LIN {X 0,Y 71.965,Z 1200.65,A -85,B 0,C 180,E1 3862.817,E2 3862.817} C_VEL
LIN {X 0,Y 71.914,Z 1200.39,A -85,B 0,C 180,E1 3872.39,E2 3872.39} C_VEL
LIN {X 0,Y 72.406,Z 1199.456,A -85,B 0,C 180,E1 3884.392,E2 3884.392} C_VEL
LIN {X 0,Y 75.878,Z 1197.57,A -85,B 0,C 180,E1 3899.18,E2 3899.18} C_VEL
LIN {X 0,Y 84.039,Z 1194.488,A -85,B 0,C 180,E1 3913.634,E2 3913.634} C_VEL
LIN {X 0,Y 99.563,Z 1189.174,A -85,B 0,C 180,E1 3927.841,E2 3927.841} C_VEL
LIN {X 0,Y 118.686,Z 1182.09,A -85,B 0,C 180,E1 3937.923,E2 3937.923} C_VEL
LIN {X 0,Y 136.218,Z 1175.067,A -85,B 0,C 180,E1 3944.061,E2 3944.061} C_VEL
LIN {X 0,Y 154.904,Z 1166.814,A -85,B 0,C 180,E1 3948.846,E2 3948.846} C_VEL
LIN {X 0,Y 178.199,Z 1155.352,A -85,B 0,C 180,E1 3953.279,E2 3953.279} C_VEL
LIN {X 0,Y 200.35,Z 1142.821,A -85,B 0,C 180,E1 3956.476,E2 3956.476} C_VEL
LIN {X 0,Y 219.029,Z 1131.127,A -85,B 0,C 180,E1 3958.647,E2 3958.647} C_VEL
LIN {X 0,Y 236.971,Z 1118.762,A -85,B 0,C 180,E1 3960.395,E2 3960.395} C_VEL
LIN {X 0,Y 256.541,Z 1103.89,A -85,B 0,C 180,E1 3962.01,E2 3962.01} C_VEL
LIN {X 0,Y 279.003,Z 1084.625,A -85,B 0,C 180,E1 3963.579,E2 3963.579} C_VEL
LIN {X 0,Y 280.373,Z 1083.351,A -85,B 0,C 180,E1 3963.668,E2 3963.668} C_VEL
LIN {X 0,Y 271.689,Z 1091.139,A -85,B 0,C 180,E1 3964.25,E2 3964.25} C_VEL
LIN {X 0,Y 266.605,Z 1095.454,A -85,B 0,C 180,E1 3964.415,E2 3964.415} C_VEL
LIN {X 0,Y 259.732,Z 1101.256,A -85,B 0,C 180,E1 3964.211,E2 3964.211} C_VEL
LIN {X 0,Y 244.077,Z 1113.399,A -85,B 0,C 180,E1 3962.959,E2 3962.959} C_VEL
LIN {X 0,Y 220.956,Z 1129.444,A -85,B 0,C 180,E1 3961.037,E2 3961.037} C_VEL
LIN {X 0,Y 201.994,Z 1141.263,A -85,B 0,C 180,E1 3959.115,E2 3959.115} C_VEL
LIN {X 0,Y 182.28,Z 1152.355,A -85,B 0,C 180,E1 3956.678,E2 3956.678} C_VEL
LIN {X 0,Y 158.208,Z 1164.433,A -85,B 0,C 180,E1 3952.849,E2 3952.849} C_VEL
LIN {X 0,Y 135.95,Z 1174.072,A -85,B 0,C 180,E1 3948.003,E2 3948.003} C_VEL
LIN {X 0,Y 117.478,Z 1181.227,A -85,B 0,C 180,E1 3942.408,E2 3942.408} C_VEL
LIN {X 0,Y 100.411,Z 1187.206,A -85,B 0,C 180,E1 3934.977,E2 3934.977} C_VEL
LIN {X 0,Y 83.535,Z 1192.691,A -85,B 0,C 180,E1 3923.315,E2 3923.315} C_VEL
LIN {X 0,Y 69.868,Z 1197.075,A -85,B 0,C 180,E1 3904.919,E2 3904.919} C_VEL
LIN {X 0,Y 64.688,Z 1199.265,A -85,B 0,C 180,E1 3887.078,E2 3887.078} C_VEL
LIN {X 0,Y 63.912,Z 1200.269,A -85,B 0,C 180,E1 3873.588,E2 3873.588} C_VEL
LIN {X 0,Y 63.942,Z 1200.51,A -85,B 0,C 180,E1 3863.716,E2 3863.716} C_VEL
LIN {X 0,Y 65.136,Z 1200.516,A -85,B 0,C 180,E1 3850.263,E2 3850.263} C_VEL
LIN {X 0,Y 71.141,Z 1199.657,A -85,B 0,C 180,E1 3832.818,E2 3832.818} C_VEL
LIN {X 0,Y 82.509,Z 1197.706,A -85,B 0,C 180,E1 3818.031,E2 3818.031} C_VEL
LIN {X 0,Y 97.644,Z 1194.686,A -85,B 0,C 180,E1 3807.018,E2 3807.018} C_VEL
LIN {X 0,Y 116.093,Z 1190.376,A -85,B 0,C 180,E1 3798.669,E2 3798.669} C_VEL
LIN {X 0,Y 140.962,Z 1183.473,A -85,B 0,C 180,E1 3791.456,E2 3791.456} C_VEL
LIN {X 0,Y 165.113,Z 1175.312,A -85,B 0,C 180,E1 3786.726,E2 3786.726} C_VEL
LIN {X 0,Y 186.353,Z 1167.079,A -85,B 0,C 180,E1 3783.661,E2 3783.661} C_VEL
LIN {X 0,Y 190.059,Z 1165.559,A -85,B 0,C 180,E1 3783.17,E2 3783.17} C_VEL
LIN {X 0,Y 167.976,Z 1174.095,A -85,B 0,C 180,E1 3780.074,E2 3780.074} C_VEL
LIN {X 0,Y 147.292,Z 1181.068,A -85,B 0,C 180,E1 3776.262,E2 3776.262} C_VEL
LIN {X 0,Y 125.611,Z 1187.374,A -85,B 0,C 180,E1 3770.762,E2 3770.762} C_VEL
LIN {X 0,Y 101.386,Z 1193.141,A -85,B 0,C 180,E1 3761.217,E2 3761.217} C_VEL
LIN {X 0,Y 85.017,Z 1196.305,A -85,B 0,C 180,E1 3750.398,E2 3750.398} C_VEL
LIN {X 0,Y 73.034,Z 1198.239,A -85,B 0,C 180,E1 3736.518,E2 3736.518} C_VEL
LIN {X 0,Y 66.274,Z 1199.108,A -85,B 0,C 180,E1 3720.686,E2 3720.686} C_VEL
LIN {X 0,Y 64.065,Z 1199.187,A -85,B 0,C 180,E1 3705.386,E2 3705.386} C_VEL
LIN {X 0,Y 63.918,Z 1198.899,A -85,B 0,C 180,E1 3694.486,E2 3694.486} C_VEL
LIN {X 0,Y 64.676,Z 1197.981,A -85,B 0,C 180,E1 3681.107,E2 3681.107} C_VEL
LIN {X 0,Y 69.216,Z 1196.076,A -85,B 0,C 180,E1 3664.319,E2 3664.319} C_VEL
LIN {X 0,Y 80.178,Z 1192.658,A -85,B 0,C 180,E1 3647.67,E2 3647.67} C_VEL
LIN {X 0,Y 99.235,Z 1186.688,A -85,B 0,C 180,E1 3633.251,E2 3633.251} C_VEL
LIN {X 0,Y 116.37,Z 1180.839,A -85,B 0,C 180,E1 3625.556,E2 3625.556} C_VEL
LIN {X 0,Y 134.074,Z 1174.148,A -85,B 0,C 180,E1 3620.009,E2 3620.009} C_VEL
LIN {X 0,Y 152.684,Z 1166.317,A -85,B 0,C 180,E1 3615.712,E2 3615.712} C_VEL
LIN {X 0,Y 175.646,Z 1155.489,A -85,B 0,C 180,E1 3611.735,E2 3611.735} C_VEL
LIN {X 0,Y 199.228,Z 1142.62,A -85,B 0,C 180,E1 3608.632,E2 3608.632} C_VEL
LIN {X 0,Y 218.421,Z 1130.906,A -85,B 0,C 180,E1 3606.612,E2 3606.612} C_VEL
LIN {X 0,Y 236.861,Z 1118.458,A -85,B 0,C 180,E1 3604.985,E2 3604.985} C_VEL
LIN {X 0,Y 253.944,Z 1105.754,A -85,B 0,C 180,E1 3603.68,E2 3603.68} C_VEL
LIN {X 0,Y 244.077,Z 1113.399,A -85,B 0,C 180,E1 3602.959,E2 3602.959} C_VEL
LIN {X 0,Y 237.846,Z 1117.949,A -85,B 0,C 180,E1 3602.729,E2 3602.729} C_VEL
LIN {X 0,Y 221.123,Z 1129.147,A -85,B 0,C 180,E1 3602.95,E2 3602.95} C_VEL
LIN {X 0,Y 214.651,Z 1133.273,A -85,B 0,C 180,E1 3602.675,E2 3602.675} C_VEL
LIN {X 0,Y 188.973,Z 1148.299,A -85,B 0,C 180,E1 3600.154,E2 3600.154} C_VEL
LIN {X 0,Y 168.131,Z 1158.981,A -85,B 0,C 180,E1 3597.538,E2 3597.538} C_VEL
LIN {X 0,Y 148.685,Z 1167.89,A -85,B 0,C 180,E1 3594.412,E2 3594.412} C_VEL
LIN {X 0,Y 128.635,Z 1176.071,A -85,B 0,C 180,E1 3590.154,E2 3590.154} C_VEL
LIN {X 0,Y 104.718,Z 1184.631,A -85,B 0,C 180,E1 3582.708,E2 3582.708} C_VEL
LIN {X 0,Y 84.953,Z 1190.695,A -85,B 0,C 180,E1 3572.676,E2 3572.676} C_VEL
LIN {X 0,Y 70.5,Z 1194.813,A -85,B 0,C 180,E1 3559.982,E2 3559.982} C_VEL
LIN {X 0,Y 60.889,Z 1197.634,A -85,B 0,C 180,E1 3543.939,E2 3543.939} C_VEL
LIN {X 0,Y 56.552,Z 1199.355,A -85,B 0,C 180,E1 3526.432,E2 3526.432} C_VEL
LIN {X 0,Y 55.914,Z 1200.217,A -85,B 0,C 180,E1 3512.049,E2 3512.049} C_VEL
LIN {X 0,Y 56.076,Z 1200.473,A -85,B 0,C 180,E1 3499.729,E2 3499.729} C_VEL
LIN {X 0,Y 59.309,Z 1200.261,A -85,B 0,C 180,E1 3480.732,E2 3480.732} C_VEL
LIN {X 0,Y 69.759,Z 1198.932,A -85,B 0,C 180,E1 3461.249,E2 3461.249} C_VEL
LIN {X 0,Y 90.166,Z 1195.477,A -85,B 0,C 180,E1 3444.591,E2 3444.591} C_VEL
LIN {X 0,Y 110.166,Z 1191.213,A -85,B 0,C 180,E1 3435.835,E2 3435.835} C_VEL
LIN {X 0,Y 130.019,Z 1186.162,A -85,B 0,C 180,E1 3430.158,E2 3430.158} C_VEL
LIN {X 0,Y 151.755,Z 1179.668,A -85,B 0,C 180,E1 3425.798,E2 3425.798} C_VEL
LIN {X 0,Y 168.931,Z 1173.751,A -85,B 0,C 180,E1 3423.16,E2 3423.16} C_VEL
LIN {X 0,Y 147.979,Z 1180.695,A -85,B 0,C 180,E1 3419.861,E2 3419.861} C_VEL
LIN {X 0,Y 126.42,Z 1186.819,A -85,B 0,C 180,E1 3415.231,E2 3415.231} C_VEL
LIN {X 0,Y 101.539,Z 1192.672,A -85,B 0,C 180,E1 3407.124,E2 3407.124} C_VEL
LIN {X 0,Y 81.149,Z 1196.331,A -85,B 0,C 180,E1 3395.751,E2 3395.751} C_VEL
LIN {X 0,Y 67.433,Z 1198.295,A -85,B 0,C 180,E1 3381.8,E2 3381.8} C_VEL
LIN {X 0,Y 59.247,Z 1199.184,A -85,B 0,C 180,E1 3365.015,E2 3365.015} C_VEL
LIN {X 0,Y 56.185,Z 1199.288,A -85,B 0,C 180,E1 3347.61,E2 3347.61} C_VEL
LIN {X 0,Y 55.918,Z 1198.999,A -85,B 0,C 180,E1 3335.13,E2 3335.13} C_VEL
LIN {X 0,Y 56.651,Z 1198.169,A -85,B 0,C 180,E1 3320.86,E2 3320.86} C_VEL
LIN {X 0,Y 60.95,Z 1196.554,A -85,B 0,C 180,E1 3303.71,E2 3303.71} C_VEL
LIN {X 0,Y 70.256,Z 1193.919,A -85,B 0,C 180,E1 3288.019,E2 3288.019} C_VEL
LIN {X 0,Y 83.774,Z 1190.178,A -85,B 0,C 180,E1 3275.748,E2 3275.748} C_VEL
LIN {X 0,Y 100.605,Z 1185.167,A -85,B 0,C 180,E1 3266.562,E2 3266.562} C_VEL
LIN {X 0,Y 123.517,Z 1177.516,A -85,B 0,C 180,E1 3258.719,E2 3258.719} C_VEL
LIN {X 0,Y 147.354,Z 1168.034,A -85,B 0,C 180,E1 3253.339,E2 3253.339} C_VEL
LIN {X 0,Y 166.592,Z 1159.398,A -85,B 0,C 180,E1 3250.167,E2 3250.167} C_VEL
LIN {X 0,Y 186.601,Z 1149.342,A -85,B 0,C 180,E1 3247.574,E2 3247.574} C_VEL
LIN {X 0,Y 209.829,Z 1136.257,A -85,B 0,C 180,E1 3245.189,E2 3245.189} C_VEL
LIN {X 0,Y 227.229,Z 1125.213,A -85,B 0,C 180,E1 3243.69,E2 3243.69} C_VEL
LIN {X 0,Y 214.651,Z 1133.273,A -85,B 0,C 180,E1 3242.675,E2 3242.675} C_VEL
LIN {X 0,Y 208.11,Z 1137.331,A -85,B 0,C 180,E1 3242.378,E2 3242.378} C_VEL
LIN {X 0,Y 189.592,Z 1147.773,A -85,B 0,C 180,E1 3242.522,E2 3242.522} C_VEL
LIN {X 0,Y 183.785,Z 1150.764,A -85,B 0,C 180,E1 3242.181,E2 3242.181} C_VEL
LIN {X 0,Y 163.976,Z 1160.546,A -85,B 0,C 180,E1 3239.922,E2 3239.922} C_VEL
LIN {X 0,Y 139.286,Z 1171.34,A -85,B 0,C 180,E1 3236.198,E2 3236.198} C_VEL
LIN {X 0,Y 114.458,Z 1180.427,A -85,B 0,C 180,E1 3230.793,E2 3230.793} C_VEL
LIN {X 0,Y 95.414,Z 1186.509,A -85,B 0,C 180,E1 3224.597,E2 3224.597} C_VEL
LIN {X 0,Y 77.874,Z 1191.456,A -85,B 0,C 180,E1 3215.727,E2 3215.727} C_VEL
LIN {X 0,Y 61.649,Z 1195.633,A -85,B 0,C 180,E1 3201.122,E2 3201.122} C_VEL
LIN {X 0,Y 50.064,Z 1198.813,A -85,B 0,C 180,E1 3176.064,E2 3176.064} C_VEL
LIN {X 0,Y 47.932,Z 1199.998,A -85,B 0,C 180,E1 3155.987,E2 3155.987} C_VEL
LIN {X 0,Y 47.918,Z 1200.25,A -85,B 0,C 180,E1 3145.212,E2 3145.212} C_VEL
LIN {X 0,Y 49.613,Z 1200.409,A -85,B 0,C 180,E1 3126.23,E2 3126.23} C_VEL
LIN {X 0,Y 58.849,Z 1199.542,A -85,B 0,C 180,E1 3103.065,E2 3103.065} C_VEL
LIN {X 0,Y 73.954,Z 1197.556,A -85,B 0,C 180,E1 3087.367,E2 3087.367} C_VEL
LIN {X 0,Y 92.135,Z 1194.501,A -85,B 0,C 180,E1 3077.257,E2 3077.257} C_VEL
LIN {X 0,Y 112.986,Z 1190.146,A -85,B 0,C 180,E1 3070.195,E2 3070.195} C_VEL
LIN {X 0,Y 139.408,Z 1183.343,A -85,B 0,C 180,E1 3064.492,E2 3064.492} C_VEL
LIN {X 0,Y 147.603,Z 1180.812,A -85,B 0,C 180,E1 3063.158,E2 3063.158} C_VEL
LIN {X 0,Y 125.994,Z 1186.779,A -85,B 0,C 180,E1 3059.2,E2 3059.2} C_VEL
LIN {X 0,Y 100.889,Z 1192.515,A -85,B 0,C 180,E1 3052.329,E2 3052.329} C_VEL
LIN {X 0,Y 77.993,Z 1196.366,A -85,B 0,C 180,E1 3041.561,E2 3041.561} C_VEL
LIN {X 0,Y 62.498,Z 1198.353,A -85,B 0,C 180,E1 3027.985,E2 3027.985} C_VEL
LIN {X 0,Y 52.181,Z 1199.284,A -85,B 0,C 180,E1 3009.222,E2 3009.222} C_VEL
LIN {X 0,Y 48.289,Z 1199.365,A -85,B 0,C 180,E1 2989.347,E2 2989.347} C_VEL
LIN {X 0,Y 47.916,Z 1199.075,A -85,B 0,C 180,E1 2974.788,E2 2974.788} C_VEL
LIN {X 0,Y 48.918,Z 1198.224,A -85,B 0,C 180,E1 2958.206,E2 2958.206} C_VEL
LIN {X 0,Y 54.283,Z 1196.588,A -85,B 0,C 180,E1 2938.953,E2 2938.953} C_VEL
LIN {X 0,Y 65.167,Z 1193.919,A -85,B 0,C 180,E1 2922.464,E2 2922.464} C_VEL
LIN {X 0,Y 80.863,Z 1189.966,A -85,B 0,C 180,E1 2910.056,E2 2910.056} C_VEL
LIN {X 0,Y 101.174,Z 1184.247,A -85,B 0,C 180,E1 2900.842,E2 2900.842} C_VEL
LIN {X 0,Y 126.644,Z 1175.714,A -85,B 0,C 180,E1 2893.812,E2 2893.812} C_VEL
LIN {X 0,Y 147.206,Z 1167.691,A -85,B 0,C 180,E1 2889.98,E2 2889.98} C_VEL
LIN {X 0,Y 167.276,Z 1158.818,A -85,B 0,C 180,E1 2887.148,E2 2887.148} C_VEL
LIN {X 0,Y 188.633,Z 1148.176,A -85,B 0,C 180,E1 2884.795,E2 2884.795} C_VEL
LIN {X 0,Y 200.192,Z 1141.797,A -85,B 0,C 180,E1 2883.723,E2 2883.723} C_VEL
LIN {X 0,Y 183.785,Z 1150.764,A -85,B 0,C 180,E1 2882.181,E2 2882.181} C_VEL
LIN {X 0,Y 176.956,Z 1154.326,A -85,B 0,C 180,E1 2881.79,E2 2881.79} C_VEL
LIN {X 0,Y 157.694,Z 1163.257,A -85,B 0,C 180,E1 2881.861,E2 2881.861} C_VEL
LIN {X 0,Y 151.662,Z 1165.78,A -85,B 0,C 180,E1 2881.42,E2 2881.42} C_VEL
LIN {X 0,Y 130.041,Z 1174.353,A -85,B 0,C 180,E1 2878.26,E2 2878.26} C_VEL
LIN {X 0,Y 109.563,Z 1181.432,A -85,B 0,C 180,E1 2874.109,E2 2874.109} C_VEL
LIN {X 0,Y 87.756,Z 1187.944,A -85,B 0,C 180,E1 2867.497,E2 2867.497} C_VEL
LIN {X 0,Y 64.203,Z 1193.815,A -85,B 0,C 180,E1 2854.589,E2 2854.589} C_VEL
LIN {X 0,Y 49.212,Z 1197.11,A -85,B 0,C 180,E1 2837.005,E2 2837.005} C_VEL
LIN {X 0,Y 41.445,Z 1199.042,A -85,B 0,C 180,E1 2814.212,E2 2814.212} C_VEL
LIN {X 0,Y 39.912,Z 1199.997,A -85,B 0,C 180,E1 2794.31,E2 2794.31} C_VEL
LIN {X 0,Y 39.993,Z 1200.193,A -85,B 0,C 180,E1 2781.373,E2 2781.373} C_VEL
LIN {X 0,Y 43.269,Z 1200.255,A -85,B 0,C 180,E1 2757.894,E2 2757.894} C_VEL
LIN {X 0,Y 54.873,Z 1199.344,A -85,B 0,C 180,E1 2734.92,E2 2734.92} C_VEL
LIN {X 0,Y 71.607,Z 1197.369,A -85,B 0,C 180,E1 2720.687,E2 2720.687} C_VEL
LIN {X 0,Y 90.923,Z 1194.328,A -85,B 0,C 180,E1 2711.843,E2 2711.843} C_VEL
LIN {X 0,Y 113.523,Z 1189.789,A -85,B 0,C 180,E1 2705.586,E2 2705.586} C_VEL
LIN {X 0,Y 125.913,Z 1186.804,A -85,B 0,C 180,E1 2703.135,E2 2703.135} C_VEL
LIN {X 0,Y 99.535,Z 1192.619,A -85,B 0,C 180,E1 2697.121,E2 2697.121} C_VEL
LIN {X 0,Y 74.815,Z 1196.513,A -85,B 0,C 180,E1 2687.317,E2 2687.317} C_VEL
LIN {X 0,Y 57.574,Z 1198.486,A -85,B 0,C 180,E1 2674.267,E2 2674.267} C_VEL
LIN {X 0,Y 45.478,Z 1199.385,A -85,B 0,C 180,E1 2654.712,E2 2654.712} C_VEL
LIN {X 0,Y 40.443,Z 1199.442,A -85,B 0,C 180,E1 2631.768,E2 2631.768} C_VEL
LIN {X 0,Y 39.918,Z 1199.174,A -85,B 0,C 180,E1 2615.75,E2 2615.75} C_VEL
LIN {X 0,Y 40.924,Z 1198.412,A -85,B 0,C 180,E1 2597.298,E2 2597.298} C_VEL
LIN {X 0,Y 47.08,Z 1196.843,A -85,B 0,C 180,E1 2575.012,E2 2575.012} C_VEL
LIN {X 0,Y 59.951,Z 1194.099,A -85,B 0,C 180,E1 2556.818,E2 2556.818} C_VEL
LIN {X 0,Y 76.29,Z 1190.359,A -85,B 0,C 180,E1 2545.27,E2 2545.27} C_VEL
LIN {X 0,Y 95.361,Z 1185.349,A -85,B 0,C 180,E1 2537.422,E2 2537.422} C_VEL
LIN {X 0,Y 120.232,Z 1177.7,A -85,B 0,C 180,E1 2531.101,E2 2531.101} C_VEL
LIN {X 0,Y 145.05,Z 1168.378,A -85,B 0,C 180,E1 2526.966,E2 2526.966} C_VEL
LIN {X 0,Y 165.48,Z 1159.584,A -85,B 0,C 180,E1 2524.472,E2 2524.472} C_VEL
LIN {X 0,Y 172.336,Z 1156.447,A -85,B 0,C 180,E1 2523.712,E2 2523.712} C_VEL
LIN {X 0,Y 151.662,Z 1165.78,A -85,B 0,C 180,E1 2521.42,E2 2521.42} C_VEL
LIN {X 0,Y 144.58,Z 1168.688,A -85,B 0,C 180,E1 2520.903,E2 2520.903} C_VEL
LIN {X 0,Y 124.697,Z 1176.178,A -85,B 0,C 180,E1 2520.834,E2 2520.834} C_VEL
LIN {X 0,Y 118.491,Z 1178.219,A -85,B 0,C 180,E1 2520.225,E2 2520.225} C_VEL
LIN {X 0,Y 93.347,Z 1185.809,A -85,B 0,C 180,E1 2514.961,E2 2514.961} C_VEL
LIN {X 0,Y 73.423,Z 1190.879,A -85,B 0,C 180,E1 2508.213,E2 2508.213} C_VEL
LIN {X 0,Y 55.242,Z 1194.799,A -85,B 0,C 180,E1 2497.378,E2 2497.378} C_VEL
LIN {X 0,Y 40.811,Z 1197.551,A -85,B 0,C 180,E1 2479.418,E2 2479.418} C_VEL
LIN {X 0,Y 33.063,Z 1199.201,A -85,B 0,C 180,E1 2453.149,E2 2453.149} C_VEL
LIN {X 0,Y 31.912,Z 1199.945,A -85,B 0,C 180,E1 2431.795,E2 2431.795} C_VEL
LIN {X 0,Y 32.502,Z 1200.176,A -85,B 0,C 180,E1 2412.083,E2 2412.083} C_VEL
LIN {X 0,Y 39.713,Z 1200.025,A -85,B 0,C 180,E1 2383.102,E2 2383.102} C_VEL
LIN {X 0,Y 55.349,Z 1198.864,A -85,B 0,C 180,E1 2362.885,E2 2362.885} C_VEL
LIN {X 0,Y 80.113,Z 1195.923,A -85,B 0,C 180,E1 2349.61,E2 2349.61} C_VEL
LIN {X 0,Y 103.727,Z 1191.744,A -85,B 0,C 180,E1 2343.093,E2 2343.093} C_VEL
LIN {X 0,Y 75.134,Z 1196.343,A -85,B 0,C 180,E1 2334.655,E2 2334.655} C_VEL
LIN {X 0,Y 54.506,Z 1198.536,A -85,B 0,C 180,E1 2322.533,E2 2322.533} C_VEL
LIN {X 0,Y 39.674,Z 1199.474,A -85,B 0,C 180,E1 2302.781,E2 2302.781} C_VEL
LIN {X 0,Y 32.694,Z 1199.519,A -85,B 0,C 180,E1 2275.351,E2 2275.351} C_VEL
LIN {X 0,Y 31.916,Z 1199.25,A -85,B 0,C 180,E1 2255.393,E2 2255.393} C_VEL
LIN {X 0,Y 33.402,Z 1198.467,A -85,B 0,C 180,E1 2232.582,E2 2232.582} C_VEL
LIN {X 0,Y 41.345,Z 1196.876,A -85,B 0,C 180,E1 2207.38,E2 2207.38} C_VEL
LIN {X 0,Y 55.486,Z 1194.266,A -85,B 0,C 180,E1 2190.123,E2 2190.123} C_VEL
LIN {X 0,Y 74.085,Z 1190.348,A -85,B 0,C 180,E1 2179.139,E2 2179.139} C_VEL
LIN {X 0,Y 95.123,Z 1185.067,A -85,B 0,C 180,E1 2172.168,E2 2172.168} C_VEL
LIN {X 0,Y 121.835,Z 1176.934,A -85,B 0,C 180,E1 2166.781,E2 2166.781} C_VEL
LIN {X 0,Y 144.053,Z 1168.764,A -85,B 0,C 180,E1 2163.739,E2 2163.739} C_VEL
LIN {X 0,Y 118.491,Z 1178.219,A -85,B 0,C 180,E1 2160.225,E2 2160.225} C_VEL
LIN {X 0,Y 111.194,Z 1180.511,A -85,B 0,C 180,E1 2159.491,E2 2159.491} C_VEL
LIN {X 0,Y 90.732,Z 1186.223,A -85,B 0,C 180,E1 2159.167,E2 2159.167} C_VEL
LIN {X 0,Y 84.443,Z 1187.839,A -85,B 0,C 180,E1 2158.231,E2 2158.231} C_VEL
LIN {X 0,Y 58.076,Z 1193.639,A -85,B 0,C 180,E1 2148.912,E2 2148.912} C_VEL
LIN {X 0,Y 39.038,Z 1196.936,A -85,B 0,C 180,E1 2133.693,E2 2133.693} C_VEL
LIN {X 0,Y 26.956,Z 1198.869,A -85,B 0,C 180,E1 2106.403,E2 2106.403} C_VEL
LIN {X 0,Y 23.911,Z 1199.823,A -85,B 0,C 180,E1 2074.797,E2 2074.797} C_VEL
LIN {X 0,Y 24.32,Z 1200.016,A -85,B 0,C 180,E1 2053.274,E2 2053.274} C_VEL
LIN {X 0,Y 31.917,Z 1200.048,A -85,B 0,C 180,E1 2018.449,E2 2018.449} C_VEL
LIN {X 0,Y 48.255,Z 1199.159,A -85,B 0,C 180,E1 1997.609,E2 1997.609} C_VEL
LIN {X 0,Y 68.499,Z 1197.184,A -85,B 0,C 180,E1 1986.987,E2 1986.987} C_VEL
LIN {X 0,Y 81.106,Z 1195.589,A -85,B 0,C 180,E1 1983.081,E2 1983.081} C_VEL
LIN {X 0,Y 54.353,Z 1198.468,A -85,B 0,C 180,E1 1972.601,E2 1972.601} C_VEL
LIN {X 0,Y 35.496,Z 1199.547,A -85,B 0,C 180,E1 1954.339,E2 1954.339} C_VEL
LIN {X 0,Y 25.436,Z 1199.621,A -85,B 0,C 180,E1 1923.39,E2 1923.39} C_VEL
LIN {X 0,Y 23.922,Z 1199.349,A -85,B 0,C 180,E1 1897.204,E2 1897.204} C_VEL
LIN {X 0,Y 25.546,Z 1198.654,A -85,B 0,C 180,E1 1869.375,E2 1869.375} C_VEL
LIN {X 0,Y 35.136,Z 1197.131,A -85,B 0,C 180,E1 1839.796,E2 1839.796} C_VEL
LIN {X 0,Y 51.903,Z 1194.434,A -85,B 0,C 180,E1 1822.383,E2 1822.383} C_VEL
LIN {X 0,Y 71.836,Z 1190.539,A -85,B 0,C 180,E1 1813.019,E2 1813.019} C_VEL
LIN {X 0,Y 92.781,Z 1185.53,A -85,B 0,C 180,E1 1807.504,E2 1807.504} C_VEL
LIN {X 0,Y 114.731,Z 1179.226,A -85,B 0,C 180,E1 1803.763,E2 1803.763} C_VEL
LIN {X 0,Y 91.986,Z 1185.852,A -85,B 0,C 180,E1 1799.93,E2 1799.93} C_VEL
LIN {X 0,Y 84.443,Z 1187.839,A -85,B 0,C 180,E1 1798.231,E2 1798.231} C_VEL
LIN {X 0,Y 77.072,Z 1189.63,A -85,B 0,C 180,E1 1797.054,E2 1797.054} C_VEL
LIN {X 0,Y 56.21,Z 1193.652,A -85,B 0,C 180,E1 1796.032,E2 1796.032} C_VEL
LIN {X 0,Y 49.833,Z 1194.692,A -85,B 0,C 180,E1 1794.225,E2 1794.225} C_VEL
LIN {X 0,Y 30.861,Z 1197.494,A -85,B 0,C 180,E1 1779.978,E2 1779.978} C_VEL
LIN {X 0,Y 18.201,Z 1199.098,A -85,B 0,C 180,E1 1747.176,E2 1747.176} C_VEL
LIN {X 0,Y 15.92,Z 1199.771,A -85,B 0,C 180,E1 1709.999,E2 1709.999} C_VEL
LIN {X 0,Y 19.223,Z 1200.035,A -85,B 0,C 180,E1 1667.455,E2 1667.455} C_VEL
LIN {X 0,Y 37.09,Z 1199.686,A -85,B 0,C 180,E1 1633.956,E2 1633.956} C_VEL
LIN {X 0,Y 57.343,Z 1198.305,A -85,B 0,C 180,E1 1622.998,E2 1622.998} C_VEL
LIN {X 0,Y 33.629,Z 1199.609,A -85,B 0,C 180,E1 1608.862,E2 1608.862} C_VEL
LIN {X 0,Y 18.863,Z 1199.716,A -85,B 0,C 180,E1 1576.439,E2 1576.439} C_VEL
LIN {X 0,Y 15.919,Z 1199.425,A -85,B 0,C 180,E1 1537.217,E2 1537.217} C_VEL
LIN {X 0,Y 18.743,Z 1198.709,A -85,B 0,C 180,E1 1497.761,E2 1497.761} C_VEL
LIN {X 0,Y 31.451,Z 1197.164,A -85,B 0,C 180,E1 1467.109,E2 1467.109} C_VEL
LIN {X 0,Y 50.332,Z 1194.445,A -85,B 0,C 180,E1 1453.248,E2 1453.248} C_VEL
LIN {X 0,Y 71.427,Z 1190.529,A -85,B 0,C 180,E1 1446.347,E2 1446.347} C_VEL
LIN {X 0,Y 83.736,Z 1187.843,A -85,B 0,C 180,E1 1443.78,E2 1443.78} C_VEL
LIN {X 0,Y 56.079,Z 1193.634,A -85,B 0,C 180,E1 1436.805,E2 1436.805} C_VEL
LIN {X 0,Y 49.833,Z 1194.692,A -85,B 0,C 180,E1 1434.225,E2 1434.225} C_VEL
LIN {X 0,Y 42.437,Z 1195.922,A -85,B 0,C 180,E1 1431.685,E2 1431.685} C_VEL
LIN {X 0,Y 19.847,Z 1198.407,A -85,B 0,C 180,E1 1425.007,E2 1425.007} C_VEL
LIN {X 0,Y 15.309,Z 1198.751,A -85,B 0,C 180,E1 1417.978,E2 1417.978} C_VEL
LIN {X 0,Y 7.919,Z 1199.65,A -85,B 0,C 180,E1 1357.253,E2 1357.253} C_VEL
LIN {X 0,Y 10.588,Z 1199.837,A -85,B 0,C 180,E1 1300.93,E2 1300.93} C_VEL
LIN {X 0,Y 26.19,Z 1199.865,A -85,B 0,C 180,E1 1266.973,E2 1266.973} C_VEL
LIN {X 0,Y 32.039,Z 1199.71,A -85,B 0,C 180,E1 1262.971,E2 1262.971} C_VEL
LIN {X 0,Y 13.449,Z 1199.788,A -85,B 0,C 180,E1 1238.177,E2 1238.177} C_VEL
LIN {X 0,Y 7.914,Z 1199.501,A -85,B 0,C 180,E1 1177.259,E2 1177.259} C_VEL
LIN {X 0,Y 13.477,Z 1198.763,A -85,B 0,C 180,E1 1115.308,E2 1115.308} C_VEL
LIN {X 0,Y 30.601,Z 1197.087,A -85,B 0,C 180,E1 1091.414,E2 1091.414} C_VEL
LIN {X 0,Y 49.623,Z 1194.533,A -85,B 0,C 180,E1 1083.813,E2 1083.813} C_VEL
LIN {X 0,Y 29.089,Z 1197.349,A -85,B 0,C 180,E1 1075.416,E2 1075.416} C_VEL
LIN {X 0,Y 15.309,Z 1198.751,A -85,B 0,C 180,E1 1057.978,E2 1057.978} C_VEL
LIN {X 0,Y 13.794,Z 1200.747,A -85,B 0,C 180,E1 1053.709,E2 1053.709} C_VEL
LIN {X 0,Y 13.794,Z 1215,A -85,B 0,C 180,E1 1053.709,E2 1053.709} C_VEL
LIN {X 0,Y 13.794,Z 1215,A -85,B 0,C 180,E1 1053.709,E2 1053.709}

QRS_NEXT_CUT()

QRS_NEXT()
QRS_HOME()

END
